{attribute 'qualified_only'}
{attribute 'strict'}
{attribute 'to_string'}
TYPE E_EM_LogicExample1_Seq_StopServos :
(
	Idle	:= c_nSeqIdle,
	Start	:= c_nSeqStart,
	
	Busy,
	
	Ready	:= c_nSeqReady,
	Error	:= c_nSeqError
);
END_TYPE

(* stored: Version 1.1.0.1, ProductVersion 3.1.4024.10
   DUT E_EM_LogicExample1_Seq_StopServos: Id {c3c967bc-8dd8-472a-af89-edf9be668910} *)
